// TIA Portal V20 export
DATA_BLOCK "DB_Traffic_Lights"   // DB1
{ S7_Optimized_Access := 'TRUE' }
// stored: MemoryReserve 100
   VAR
      Process_Step : Int;
      Process_Start : Bool;
      "Timer" : IEC_TIMER;
      "Counter" { S7_SetPoint := 'True'} : IEC_COUNTER;
   END_VAR
   VAR RETAIN
      Positive_Edge { S7_SetPoint := 'True'} : Bool;
   END_VAR
   VAR
      Timer2 : IEC_TIMER;
   END_VAR
BEGIN
END_DATA_BLOCK
